// TIA Portal V17 export
// export: Created 2026-04-13T11:12:44.9371969Z, ExportSetting WithDefaults, DisplayName Totally Integrated Automation Portal, DisplayVersion V17 Update 4, DisplayName TIA Portal Openness, DisplayVersion V17 Update 4, DisplayName TIA Portal Version Control Interface, DisplayVersion V17, DisplayName SINAMICS Startdrive Advanced, DisplayVersion V17, DisplayName SINAMICS Startdrive G130, G150, S120, S150, SINAMICS MV, S210, DisplayVersion V17, DisplayName SINAMICS Startdrive G110M, G120, G120C, G120D, G120P, G115D, DisplayVersion V17, DisplayName STEP 7 Professional, DisplayVersion V17 Update 4, DisplayName STEP 7 Safety, DisplayVersion V17, DisplayName WinCC Professional, DisplayVersion V17 Update 4
FUNCTION_BLOCK "Send_P2P"   // FB613, SCL
TITLE = Send data
AUTHOR : SIMATIC
FAMILY : Freeport
NAME : SendP2P
VERSION : 4.0
// stored: IsIECCheckEnabled true, SetENOAutomatically false, UDAEnableTagReadback false
   VAR_INPUT
      REQ : Bool;   // Startet die angeforderte Übertragung bei steigender Flanke / Activates the requested transmission on rising edge
      PORT : PORT := 16#0000;   // Kommunikationsport, Hardwarekennung / Communication port, Hardware Identifier
      BUFFER : Variant;   // Referenz auf den Sendepuffer / Reference to the send buffer
      LENGTH : UInt := 0;   // Übertragene Datenlänge in Byte / Transmitted frame length in bytes
   END_VAR
   VAR_OUTPUT
      UNIVERSAL : Bool;   // Access mode of communication module. 0 = universal, 1 = performance
      DONE : Bool;   // Anweisung beendet ohne Fehler / Instruction finished without error
      ERROR : Bool;   // Anweisung beendet mit Fehler / Instruction finished with error
      STATUS : Word := W#16#7000;   // Zusätzliche Fehlerinformation / Detailed error information
   END_VAR
   VAR
      OldPORT : PORT := 16#0000;   // Nur für internen Gebrauch / Save value for Communication port
      send_length : UInt;   // Übertragene Datenlänge in Byte / For internal use only
      max_record_len : UInt := 1026;   // Nur für internen Gebrauch / For internal use only
      max_telegram_len : UInt;
      b_e_REQ : Bool;   // Flankenbit für REQ / Edge flag for REQ
      isClassic : Bool;   // Nur für internen Gebrauch / For internal use only
      first_sent : Bool;
      y_state : SInt := 0;   // Status der Anweisung / State of instruction
      y_nr_rec : SInt;   // Nur für internen Gebrauch / Sequence number of data records
      ser_nr_old : USInt;
      ser_nr : USInt;   // Nur für internen Gebrauch / For internal use only
      module_initialized { ExternalAccessible := 'False'; ExternalVisible := 'False'; ExternalWritable := 'False'} : Bool;
   END_VAR
   VAR DB_SPECIFIC
      SendBuffer : Array[0..1026] of Byte;   // Nur für internen Gebrauch / For internal use only
   END_VAR
   VAR
      i_addr : UDInt;   // IO Adresse des Moduls / IO address of the module
      o_addr { ExternalAccessible := 'False'; ExternalVisible := 'False'; ExternalWritable := 'False'} : UDInt;
      WRREC { S7_SetPoint := 'True'} : WRREC;   // Lokale Instanz der Anweisung WRREC / Local instance of instruction WRREC
      PTP_STATUS { S7_SetPoint := 'True'} : P2P_SendGetData;   // Nur für internen Gebrauch / For internal use only
      InitTimeout { ExternalAccessible := 'False'; ExternalVisible := 'False'; ExternalWritable := 'False'; S7_SetPoint := 'True'} : TON_TIME;
   END_VAR
BEGIN
END_FUNCTION_BLOCK
